SUBAPPLICATION Uebung_010f2_AX (* AuxFunction2_X1 auf DigitalOutput_Q1 mit GreenWhiteBackground mit Subapp *)
  (* Standard: 61499-2; Description: Copyright (c) 2026 Meisterschulen am Ostbahnhof This program and the accompanying materials are made available under the terms of the Eclipse Public License 2.0 which is available at https://www.eclipse.org/legal/epl-2.0/ SPDX-License-Identifier: EPL-2.0 *)
  (* Version 1.0, 2026-09-06, Franz Höpfinger, Meisterschulen am Ostbahnhof, initial API and implementation and/or initial documentation *)
  PACKAGE Uebungen;
  IMPORT Uebungen::const::UT::DefaultPool::AuxFunction2_X1;
  IMPORT logiBUS::io::DQ::logiBUS_DO;
  (* Documentation:
  AuxFunction2_X1 auf DigitalOutput_Q1 mit GreenWhiteBackground mit Subapp
   Löst den in Uebung_010f_AX notierten Nachteil auf, genau wie Uebung_010c2_AX es für Uebung_010c_AX tut: die Object-ID wird nicht mehr an zwei Stellen (Aux-FB und GreenWhiteBackground2_AX) einzeln eingetragen, sondern nur noch einmal, als Parameter der gekapselten Subapp Uebung_10f2_sub_AX.
   Funktionsbeschreibung
    - Die Subapp exponiert u16ObjIdA und Output als einzige Eingänge nach außen.
   - Intern verteilt eine DataConnection von u16ObjIdA auf sowohl AuxFunction2_X1.u16ObjId als auch GreenWhiteBackground2_AX.u16ObjIdA - der Wert muss beim Aufruf der Subapp nur noch einmal angegeben werden.
   - AX_SPLIT_2 und GreenWhiteBackground2_AX selbst bleiben unverändert gegenüber Uebung_010f_AX: die AUX-Farbe geht weiterhin sowohl an den VT-Bildschirm als auch an das Aux-Handle - das ist kein Nachteil, sondern notwendig, und wird hier nicht wegoptimiert.
  *)
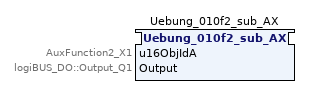
  SUBAPPS
    Uebung_010f2_sub_AX : Uebungen::Uebung_010f2_sub_AX(u16ObjIdA := AuxFunction2_X1 (* Object ID AUX *), Output := logiBUS_DO::Output_Q1 (* Identify the Output Output_Q1..Q8 *));
  END_SUBAPPS
END_SUBAPPLICATION
